KUKA KRL program: PROTON_EXHIBITION_CHECK.src

&ACCESS RVP
&REL 2
&PARAM DISKPATH = KRC:\\R1\\Program
DEF PROTON_EXHIBITION_CHECK()
   BAS(#INITMOV, 0)

   \
       ;FOLD SPTP P1 Vel=100 % PDAT1 Tool[1]:Tool Base[0] ;%{PE}
       ;FOLD Parameters ;%{h}
       ;Params IlfProvider=kukaroboter.basistech.inlineforms.movement.spline; Kuka.IsGlobalPoint=False; Kuka.PointName=P1; Kuka.BlendingEnabled=False; Kuka.MoveDataPtpName=PDAT1; Kuka.VelocityPtp=100; Kuka.VelocityFieldEnabled=True; Kuka.ColDetectFieldEnabled=True; Kuka.CurrentCDSetIndex=0; Kuka.MovementParameterFieldEnabled=True; IlfCommand=SPTP
       ;ENDFOLD
       SPTP XP1 WITH $VEL_AXIS[1] = SVEL_JOINT(100.0), $TOOL = STOOL2(FP1), $BASE = SBASE(FP1.BASE_NO), $IPO_MODE = SIPO_MODE(FP1.IPO_FRAME), $LOAD = SLOAD(FP1.TOOL_NO), $ACC_AXIS[1] = SACC_JOINT(PPDAT1), $APO = SAPO_PTP(PPDAT1), $GEAR_JERK[1] = SGEAR_JERK(PPDAT1), $COLLMON_TOL_PRO[1] = USE_CM_PRO_VALUES(0)
       ;ENDFOLD

   \
       ;FOLD SPTP P2 Vel=100 % PDAT2 Tool[1]:Tool Base[0] ;%{PE}
       ;FOLD Parameters ;%{h}
       ;Params IlfProvider=kukaroboter.basistech.inlineforms.movement.spline; Kuka.IsGlobalPoint=False; Kuka.PointName=P2; Kuka.BlendingEnabled=False; Kuka.MoveDataPtpName=PDAT2; Kuka.VelocityPtp=100; Kuka.VelocityFieldEnabled=True; Kuka.ColDetectFieldEnabled=True; Kuka.CurrentCDSetIndex=0; Kuka.MovementParameterFieldEnabled=True; IlfCommand=SPTP
       ;ENDFOLD
       SPTP XP2 WITH $VEL_AXIS[1] = SVEL_JOINT(100.0), $TOOL = STOOL2(FP2), $BASE = SBASE(FP2.BASE_NO), $IPO_MODE = SIPO_MODE(FP2.IPO_FRAME), $LOAD = SLOAD(FP2.TOOL_NO), $ACC_AXIS[1] = SACC_JOINT(PPDAT2), $APO = SAPO_PTP(PPDAT2), $GEAR_JERK[1] = SGEAR_JERK(PPDAT2), $COLLMON_TOL_PRO[1] = USE_CM_PRO_VALUES(0)
       ;ENDFOLD

   \
       ;FOLD SPTP P3 Vel=100 % PDAT3 Tool[1]:Tool Base[0] ;%{PE}
       ;FOLD Parameters ;%{h}
       ;Params IlfProvider=kukaroboter.basistech.inlineforms.movement.spline; Kuka.IsGlobalPoint=False; Kuka.PointName=P3; Kuka.BlendingEnabled=False; Kuka.MoveDataPtpName=PDAT3; Kuka.VelocityPtp=100; Kuka.VelocityFieldEnabled=True; Kuka.ColDetectFieldEnabled=True; Kuka.CurrentCDSetIndex=0; Kuka.MovementParameterFieldEnabled=True; IlfCommand=SPTP
       ;ENDFOLD
       SPTP XP3 WITH $VEL_AXIS[1] = SVEL_JOINT(100.0), $TOOL = STOOL2(FP3), $BASE = SBASE(FP3.BASE_NO), $IPO_MODE = SIPO_MODE(FP3.IPO_FRAME), $LOAD = SLOAD(FP3.TOOL_NO), $ACC_AXIS[1] = SACC_JOINT(PPDAT3), $APO = SAPO_PTP(PPDAT3), $GEAR_JERK[1] = SGEAR_JERK(PPDAT3), $COLLMON_TOL_PRO[1] = USE_CM_PRO_VALUES(0)
       ;ENDFOLD

   \
       ;FOLD SPTP P4 Vel=100 % PDAT4 Tool[1]:Tool Base[0] ;%{PE}
       ;FOLD Parameters ;%{h}
       ;Params IlfProvider=kukaroboter.basistech.inlineforms.movement.spline; Kuka.IsGlobalPoint=False; Kuka.PointName=P4; Kuka.BlendingEnabled=False; Kuka.MoveDataPtpName=PDAT4; Kuka.VelocityPtp=100; Kuka.VelocityFieldEnabled=True; Kuka.ColDetectFieldEnabled=True; Kuka.CurrentCDSetIndex=0; Kuka.MovementParameterFieldEnabled=True; IlfCommand=SPTP
       ;ENDFOLD
       SPTP XP4 WITH $VEL_AXIS[1] = SVEL_JOINT(100.0), $TOOL = STOOL2(FP4), $BASE = SBASE(FP4.BASE_NO), $IPO_MODE = SIPO_MODE(FP4.IPO_FRAME), $LOAD = SLOAD(FP4.TOOL_NO), $ACC_AXIS[1] = SACC_JOINT(PPDAT4), $APO = SAPO_PTP(PPDAT4), $GEAR_JERK[1] = SGEAR_JERK(PPDAT4), $COLLMON_TOL_PRO[1] = USE_CM_PRO_VALUES(0)
       ;ENDFOLD

   \
       ;FOLD SPTP P5 Vel=100 % PDAT5 Tool[1]:Tool Base[0] ;%{PE}
       ;FOLD Parameters ;%{h}
       ;Params IlfProvider=kukaroboter.basistech.inlineforms.movement.spline; Kuka.IsGlobalPoint=False; Kuka.PointName=P5; Kuka.BlendingEnabled=False; Kuka.MoveDataPtpName=PDAT5; Kuka.VelocityPtp=100; Kuka.VelocityFieldEnabled=True; Kuka.ColDetectFieldEnabled=True; Kuka.CurrentCDSetIndex=0; Kuka.MovementParameterFieldEnabled=True; IlfCommand=SPTP
       ;ENDFOLD
       SPTP XP5 WITH $VEL_AXIS[1] = SVEL_JOINT(100.0), $TOOL = STOOL2(FP5), $BASE = SBASE(FP5.BASE_NO), $IPO_MODE = SIPO_MODE(FP5.IPO_FRAME), $LOAD = SLOAD(FP5.TOOL_NO), $ACC_AXIS[1] = SACC_JOINT(PPDAT5), $APO = SAPO_PTP(PPDAT5), $GEAR_JERK[1] = SGEAR_JERK(PPDAT5), $COLLMON_TOL_PRO[1] = USE_CM_PRO_VALUES(0)
       ;ENDFOLD

   \
       ;FOLD SPTP P6 Vel=100 % PDAT6 Tool[1]:Tool Base[0] ;%{PE}
       ;FOLD Parameters ;%{h}
       ;Params IlfProvider=kukaroboter.basistech.inlineforms.movement.spline; Kuka.IsGlobalPoint=False; Kuka.PointName=P6; Kuka.BlendingEnabled=False; Kuka.MoveDataPtpName=PDAT6; Kuka.VelocityPtp=100; Kuka.VelocityFieldEnabled=True; Kuka.ColDetectFieldEnabled=True; Kuka.CurrentCDSetIndex=0; Kuka.MovementParameterFieldEnabled=True; IlfCommand=SPTP
       ;ENDFOLD
       SPTP XP6 WITH $VEL_AXIS[1] = SVEL_JOINT(100.0), $TOOL = STOOL2(FP6), $BASE = SBASE(FP6.BASE_NO), $IPO_MODE = SIPO_MODE(FP6.IPO_FRAME), $LOAD = SLOAD(FP6.TOOL_NO), $ACC_AXIS[1] = SACC_JOINT(PPDAT6), $APO = SAPO_PTP(PPDAT6), $GEAR_JERK[1] = SGEAR_JERK(PPDAT6), $COLLMON_TOL_PRO[1] = USE_CM_PRO_VALUES(0)
       ;ENDFOLD

   \
       ;FOLD SPTP P7 Vel=100 % PDAT7 Tool[1]:Tool Base[0] ;%{PE}
       ;FOLD Parameters ;%{h}
       ;Params IlfProvider=kukaroboter.basistech.inlineforms.movement.spline; Kuka.IsGlobalPoint=False; Kuka.PointName=P7; Kuka.BlendingEnabled=False; Kuka.MoveDataPtpName=PDAT7; Kuka.VelocityPtp=100; Kuka.VelocityFieldEnabled=True; Kuka.ColDetectFieldEnabled=True; Kuka.CurrentCDSetIndex=0; Kuka.MovementParameterFieldEnabled=True; IlfCommand=SPTP
       ;ENDFOLD
       SPTP XP7 WITH $VEL_AXIS[1] = SVEL_JOINT(100.0), $TOOL = STOOL2(FP7), $BASE = SBASE(FP7.BASE_NO), $IPO_MODE = SIPO_MODE(FP7.IPO_FRAME), $LOAD = SLOAD(FP7.TOOL_NO), $ACC_AXIS[1] = SACC_JOINT(PPDAT7), $APO = SAPO_PTP(PPDAT7), $GEAR_JERK[1] = SGEAR_JERK(PPDAT7), $COLLMON_TOL_PRO[1] = USE_CM_PRO_VALUES(0)
       ;ENDFOLD

   \
       ;FOLD SPTP P8 Vel=100 % PDAT8 Tool[1]:Tool Base[0] ;%{PE}
       ;FOLD Parameters ;%{h}
       ;Params IlfProvider=kukaroboter.basistech.inlineforms.movement.spline; Kuka.IsGlobalPoint=False; Kuka.PointName=P8; Kuka.BlendingEnabled=False; Kuka.MoveDataPtpName=PDAT8; Kuka.VelocityPtp=100; Kuka.VelocityFieldEnabled=True; Kuka.ColDetectFieldEnabled=True; Kuka.CurrentCDSetIndex=0; Kuka.MovementParameterFieldEnabled=True; IlfCommand=SPTP
       ;ENDFOLD
       SPTP XP8 WITH $VEL_AXIS[1] = SVEL_JOINT(100.0), $TOOL = STOOL2(FP8), $BASE = SBASE(FP8.BASE_NO), $IPO_MODE = SIPO_MODE(FP8.IPO_FRAME), $LOAD = SLOAD(FP8.TOOL_NO), $ACC_AXIS[1] = SACC_JOINT(PPDAT8), $APO = SAPO_PTP(PPDAT8), $GEAR_JERK[1] = SGEAR_JERK(PPDAT8), $COLLMON_TOL_PRO[1] = USE_CM_PRO_VALUES(0)
       ;ENDFOLD

   \
       ;FOLD SPTP P9 Vel=100 % PDAT9 Tool[1]:Tool Base[0] ;%{PE}
       ;FOLD Parameters ;%{h}
       ;Params IlfProvider=kukaroboter.basistech.inlineforms.movement.spline; Kuka.IsGlobalPoint=False; Kuka.PointName=P9; Kuka.BlendingEnabled=False; Kuka.MoveDataPtpName=PDAT9; Kuka.VelocityPtp=100; Kuka.VelocityFieldEnabled=True; Kuka.ColDetectFieldEnabled=True; Kuka.CurrentCDSetIndex=0; Kuka.MovementParameterFieldEnabled=True; IlfCommand=SPTP
       ;ENDFOLD
       SPTP XP9 WITH $VEL_AXIS[1] = SVEL_JOINT(100.0), $TOOL = STOOL2(FP9), $BASE = SBASE(FP9.BASE_NO), $IPO_MODE = SIPO_MODE(FP9.IPO_FRAME), $LOAD = SLOAD(FP9.TOOL_NO), $ACC_AXIS[1] = SACC_JOINT(PPDAT9), $APO = SAPO_PTP(PPDAT9), $GEAR_JERK[1] = SGEAR_JERK(PPDAT9), $COLLMON_TOL_PRO[1] = USE_CM_PRO_VALUES(0)
       ;ENDFOLD

   \
       ;FOLD SPTP P10 Vel=100 % PDAT10 Tool[1]:Tool Base[0] ;%{PE}
       ;FOLD Parameters ;%{h}
       ;Params IlfProvider=kukaroboter.basistech.inlineforms.movement.spline; Kuka.IsGlobalPoint=False; Kuka.PointName=P10; Kuka.BlendingEnabled=False; Kuka.MoveDataPtpName=PDAT10; Kuka.VelocityPtp=100; Kuka.VelocityFieldEnabled=True; Kuka.ColDetectFieldEnabled=True; Kuka.CurrentCDSetIndex=0; Kuka.MovementParameterFieldEnabled=True; IlfCommand=SPTP
       ;ENDFOLD
       SPTP XP10 WITH $VEL_AXIS[1] = SVEL_JOINT(100.0), $TOOL = STOOL2(FP10), $BASE = SBASE(FP10.BASE_NO), $IPO_MODE = SIPO_MODE(FP10.IPO_FRAME), $LOAD = SLOAD(FP10.TOOL_NO), $ACC_AXIS[1] = SACC_JOINT(PPDAT10), $APO = SAPO_PTP(PPDAT10), $GEAR_JERK[1] = SGEAR_JERK(PPDAT10), $COLLMON_TOL_PRO[1] = USE_CM_PRO_VALUES(0)
       ;ENDFOLD

   \
       ;FOLD SPTP P11 Vel=100 % PDAT11 Tool[1]:Tool Base[0] ;%{PE}
       ;FOLD Parameters ;%{h}
       ;Params IlfProvider=kukaroboter.basistech.inlineforms.movement.spline; Kuka.IsGlobalPoint=False; Kuka.PointName=P11; Kuka.BlendingEnabled=False; Kuka.MoveDataPtpName=PDAT11; Kuka.VelocityPtp=100; Kuka.VelocityFieldEnabled=True; Kuka.ColDetectFieldEnabled=True; Kuka.CurrentCDSetIndex=0; Kuka.MovementParameterFieldEnabled=True; IlfCommand=SPTP
       ;ENDFOLD
       SPTP XP11 WITH $VEL_AXIS[1] = SVEL_JOINT(100.0), $TOOL = STOOL2(FP11), $BASE = SBASE(FP11.BASE_NO), $IPO_MODE = SIPO_MODE(FP11.IPO_FRAME), $LOAD = SLOAD(FP11.TOOL_NO), $ACC_AXIS[1] = SACC_JOINT(PPDAT11), $APO = SAPO_PTP(PPDAT11), $GEAR_JERK[1] = SGEAR_JERK(PPDAT11), $COLLMON_TOL_PRO[1] = USE_CM_PRO_VALUES(0)
       ;ENDFOLD

   \
       ;FOLD SPTP P12 Vel=100 % PDAT12 Tool[1]:Tool Base[0] ;%{PE}
       ;FOLD Parameters ;%{h}
       ;Params IlfProvider=kukaroboter.basistech.inlineforms.movement.spline; Kuka.IsGlobalPoint=False; Kuka.PointName=P12; Kuka.BlendingEnabled=False; Kuka.MoveDataPtpName=PDAT12; Kuka.VelocityPtp=100; Kuka.VelocityFieldEnabled=True; Kuka.ColDetectFieldEnabled=True; Kuka.CurrentCDSetIndex=0; Kuka.MovementParameterFieldEnabled=True; IlfCommand=SPTP
       ;ENDFOLD
       SPTP XP12 WITH $VEL_AXIS[1] = SVEL_JOINT(100.0), $TOOL = STOOL2(FP12), $BASE = SBASE(FP12.BASE_NO), $IPO_MODE = SIPO_MODE(FP12.IPO_FRAME), $LOAD = SLOAD(FP12.TOOL_NO), $ACC_AXIS[1] = SACC_JOINT(PPDAT12), $APO = SAPO_PTP(PPDAT12), $GEAR_JERK[1] = SGEAR_JERK(PPDAT12), $COLLMON_TOL_PRO[1] = USE_CM_PRO_VALUES(0)
       ;ENDFOLD

   \
       ;FOLD SPTP P13 Vel=100 % PDAT13 Tool[1]:Tool Base[0] ;%{PE}
       ;FOLD Parameters ;%{h}
       ;Params IlfProvider=kukaroboter.basistech.inlineforms.movement.spline; Kuka.IsGlobalPoint=False; Kuka.PointName=P13; Kuka.BlendingEnabled=False; Kuka.MoveDataPtpName=PDAT13; Kuka.VelocityPtp=100; Kuka.VelocityFieldEnabled=True; Kuka.ColDetectFieldEnabled=True; Kuka.CurrentCDSetIndex=0; Kuka.MovementParameterFieldEnabled=True; IlfCommand=SPTP
       ;ENDFOLD
       SPTP XP13 WITH $VEL_AXIS[1] = SVEL_JOINT(100.0), $TOOL = STOOL2(FP13), $BASE = SBASE(FP13.BASE_NO), $IPO_MODE = SIPO_MODE(FP13.IPO_FRAME), $LOAD = SLOAD(FP13.TOOL_NO), $ACC_AXIS[1] = SACC_JOINT(PPDAT13), $APO = SAPO_PTP(PPDAT13), $GEAR_JERK[1] = SGEAR_JERK(PPDAT13), $COLLMON_TOL_PRO[1] = USE_CM_PRO_VALUES(0)
       ;ENDFOLD

END
